// TIA Portal V20 export
TYPE "typeEmHomedCheck"
// stored: Access Published, Namespace Unit1.Em3
   STRUCT
      cmMasterVirtualAxis : Bool;
      cmDancerUnit : Bool;
      cmLoadCellAnalogInput : Bool;
      cmWebGuideEpc : Bool;
   END_STRUCT;
END_TYPE
